(* CoDeSys 2.3.9.41 project: Main.pro *)
(* Libraries: STANDARD.LIB 4.10.05 11:14:46, IECSFC.LIB 13.4.06 15:51:28, ANALYZATION.LIB 5.10.99 09:05:06, Util.lib 18.5.10 15:14:28 *)

(* PLC configuration (modules and I/O channels)
I0 AT %IX0.0 [BitInput] Discrete input 1 {ChannellName = Enter name}
I1 AT %IX0.1 [BitInput] Discrete input 2 {ChannellName = Enter name}
I2 AT %IX0.2 [BitInput] Discrete input 3 {ChannellName = Enter name}
I3 AT %IX0.3 [BitInput] Discrete input 4 {ChannellName = Enter name}
AT %IB1.0 [ByteInput] 8 discrete inputs {ChannellName = Enter name}
AT %IB1.1 [ByteInput] 4 discrete inputs {ChannellName = Enter name}
Q0 AT %QX2.0 [BitOutput] Fast discrete output 1 {ChannellName = Enter name}
AT %QX2.1 [BitOutput] Fast discrete output 2 {ChannellName = Enter name}
AT %QX2.2 [BitOutput] Fast discrete output 3 {ChannellName = Enter name}
AT %QX2.3 [BitOutput] Fast discrete output 4 {ChannellName = Enter name}
AT %QB3.0 [ByteOutput] 8 discrete outputs {ChannellName = Enter name}
AT %QB3.1 [ByteOutput] 8 discrete outputs {ChannellName = Enter name}
AT %IR4.0 [FloatInputP] You need to reboot PLC after change AI configuration! {ChannellName = Fast analog input; AIN_TYPE = 4-20 mA; Peak_Filtr = 200; Flt_Ch = Off; TauRC = 10; MinFV = 0; MaxFV = 20000.0}
AT %IR4.1 [FloatInputP] You need to reboot PLC after change AI configuration! {ChannellName = Fast analog input; AIN_TYPE = 4-20 mA; Peak_Filtr = 200; Flt_Ch = Off; TauRC = 10; MinFV = 0; MaxFV = 20000.0}
AT %IR4.2 [FloatInputP] You need to reboot PLC after change AI configuration! {ChannellName = Fast analog input; AIN_TYPE = 4-20 mA; Peak_Filtr = 200; Flt_Ch = Off; TauRC = 10; MinFV = 0; MaxFV = 20000.0}
AT %IR4.3 [FloatInputP] You need to reboot PLC after change AI configuration! {ChannellName = Fast analog input; AIN_TYPE = 4-20 mA; Peak_Filtr = 200; Flt_Ch = Off; TauRC = 10; MinFV = 0; MaxFV = 20000.0}
AT %IR4.4 [FloatInputP] You need to reboot PLC after change AI configuration! {ChannellName = Fast analog input; AIN_TYPE = 4-20 mA; Peak_Filtr = 200; Flt_Ch = Off; TauRC = 10; MinFV = 0; MaxFV = 20000.0}
AT %IR4.5 [FloatInputP] You need to reboot PLC after change AI configuration! {ChannellName = Fast analog input; AIN_TYPE = 4-20 mA; Peak_Filtr = 200; Flt_Ch = Off; TauRC = 10; MinFV = 0; MaxFV = 20000.0}
AT %IR4.6 [FloatInputP] You need to reboot PLC after change AI configuration! {ChannellName = Fast analog input; AIN_TYPE = 4-20 mA; Peak_Filtr = 200; Flt_Ch = Off; TauRC = 10; MinFV = 0; MaxFV = 20000.0}
AT %IR4.7 [FloatInputP] You need to reboot PLC after change AI configuration! {ChannellName = Fast analog input; AIN_TYPE = 4-20 mA; Peak_Filtr = 200; Flt_Ch = Off; TauRC = 10; MinFV = 0; MaxFV = 20000.0}
AT %IW4.8 [WordInput] AI read time (10ms) {ChannellName = Enter name}
Analog outputs [ID126] node 5, in %IB5 out %QB5 {ChannellName = Analog outputs}
  AT %QR5.0 [FloatOutputP] AO #1 {ChannellName = Analog output; AOUT_TYPE = 4-20 mA; SafeValueREAL = 0.0}
  AT %QR5.1 [FloatOutputP] AO #2 {ChannellName = Analog output; AOUT_TYPE = 4-20 mA; SafeValueREAL = 0.0}
  AT %QR5.2 [FloatOutputP] AO #3 {ChannellName = Analog output; AOUT_TYPE = 4-20 mA; SafeValueREAL = 0.0}
  AT %QR5.3 [FloatOutputP] AO #4 {ChannellName = Analog output; AOUT_TYPE = 4-20 mA; SafeValueREAL = 0.0}
Special input [ID103] node 6, in %IB6 out %QB6 {ChannellName = Special input}
  AT %IX6.0 [BitInput] Special input {ChannellName = Enter name}
Special output [ID104] node 7, in %IB7 out %QB7 {ChannellName = Special output}
  AT %QX7.0 [BitOutput] Special output {ChannellName = Enter name}
*)

(* POU PLC_PRG, FBD *)
PROGRAM PLC_PRG
VAR
	START: BOOL:= FALSE;
	DEC_TO_BIN: DEC_TO_BIN;
	START_RS: RS;
	DTB: DEC_TO_BIN;
	SEND: BOOL := FALSE;
	POSITION: DWORD;
	SENDING: BOOL;
	SENDING_TIMER: TOF;
	INSTRUCTION: ARRAY [1..7] OF DWORD:= 0,14,17,15,7,9,7 11,12,10, 7, 3, 4, 2, 18, 21, 19, 7, 9, 7, 11,12,10, 7, 3, 4, 2, 22, 25, 23, 7, 9, 7, 11,12,10, 7, 3, 4, 2, 26, 29, 27, 7, 9, 7, 11,12,10, 7, 3, 4, 2, 0;
	POSITION_INDEX: INT:=1;

	RESET: BOOL;
END_VAR
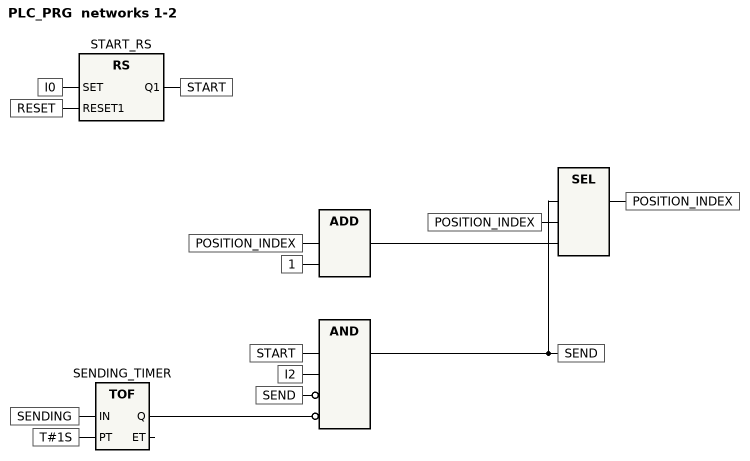
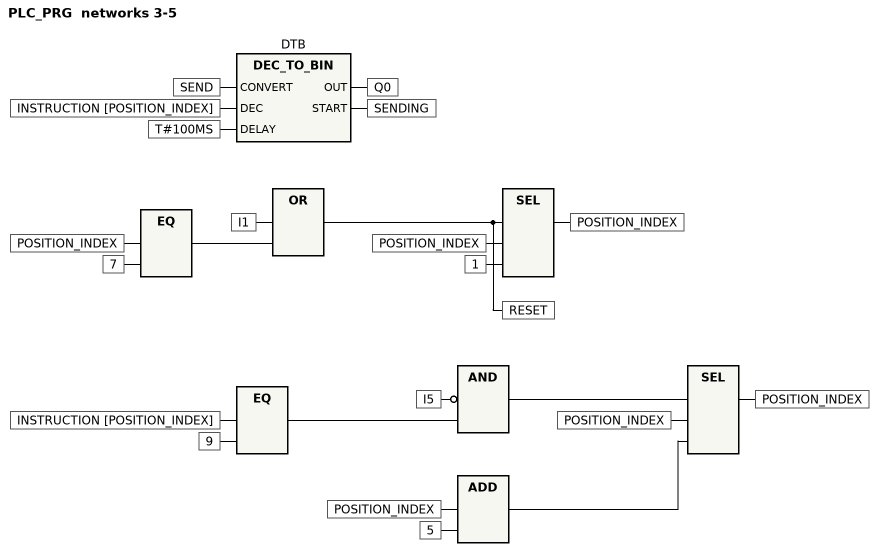
_FBD_ (* Function Block Diagram *)
NETWORK 1
	START_RS:RS(SET: I0, RESET1: RESET) => START
NETWORK 2
	SEL(<AND(START, I2, NOT SEND, NOT SENDING_TIMER:TOF(IN: SENDING, PT: T#1S)) => SEND>, POSITION_INDEX, ADD(POSITION_INDEX, 1)) => POSITION_INDEX
NETWORK 3
	DTB:DEC_TO_BIN(CONVERT: SEND, DEC: INSTRUCTION [POSITION_INDEX], DELAY: T#100MS, START => SENDING) => Q0
NETWORK 4
	SEL(<OR(I1, EQ(POSITION_INDEX, 7)) => RESET>, POSITION_INDEX, 1) => POSITION_INDEX
NETWORK 5
	SEL(AND(NOT I5, EQ(INSTRUCTION [POSITION_INDEX], 9)), POSITION_INDEX, ADD(POSITION_INDEX, 5)) => POSITION_INDEX
_END_FBD_
(* the same logic as Structured Text *)
(* Network 1 *)
START_RS(SET := I0, RESET1 := RESET);
START := START_RS.Q1;
(* Network 2 *)
SENDING_TIMER(IN := SENDING, PT := T#1S);
SEND := START AND I2 AND NOT SEND AND NOT SENDING_TIMER.Q;
POSITION_INDEX := SEL(SEND, POSITION_INDEX, POSITION_INDEX + 1);
(* Network 3 *)
DTB(CONVERT := SEND, DEC := INSTRUCTION [POSITION_INDEX], DELAY := T#100MS);
SENDING := DTB.START;
Q0 := DTB.OUT;
(* Network 4 *)
RESET := I1 OR (POSITION_INDEX = 7);
POSITION_INDEX := SEL(RESET, POSITION_INDEX, 1);
(* Network 5 *)
POSITION_INDEX := SEL(NOT I5 AND ((INSTRUCTION [POSITION_INDEX]) = 9), POSITION_INDEX, POSITION_INDEX + 5);
END_PROGRAM

(* POU DEC_TO_BIN, FBD *)
FUNCTION_BLOCK DEC_TO_BIN
VAR_INPUT
	CONVERT :BOOL :=FALSE;
	DEC :DWORD := 0;
	DELAY: TIME:= T#100MS;
END_VAR
VAR_OUTPUT
	OUT : BOOL :=FALSE;
	START : BOOL :=FALSE;
END_VAR
VAR
	RESET: BOOL :=FALSE;
	Q0, Q1,Q2,Q3,Q4,Q5,Q6,Q7,Q8,Q9,Q10: BOOL :=FALSE;
	TIMER0: TON;
	B, B0, B1,B2,B3: BOOL :=FALSE;
	TIMER6: TON;
	SETTER: RS;
	TIMER: TON;
	SETTER1: RS;
	SETTER0: RS;
	SETTER2: RS;
	SETTER3: RS;
	SETTER4: RS;
	TIMER1: TON;
	TIMER2: TON;
	TIMER3: TON;
	TIMER4: TON;
	RESET0: RS;
	TIMER5: TON;
	TIMER7: TON;
	TIMER8: TON;
	TIMER9: TON;
END_VAR
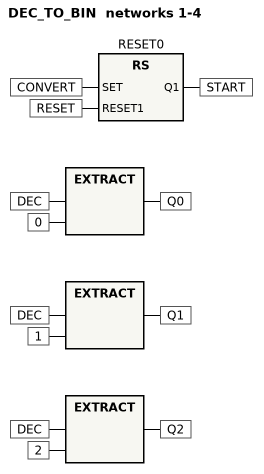
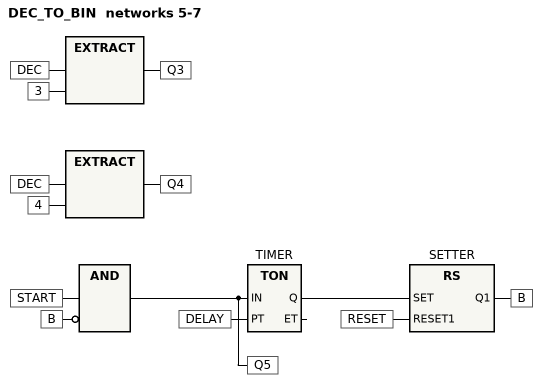
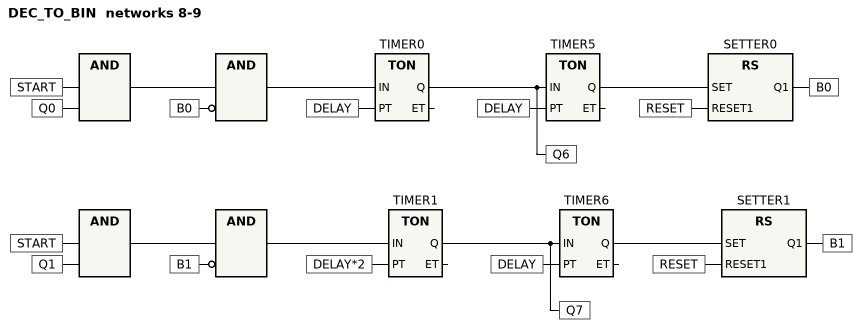
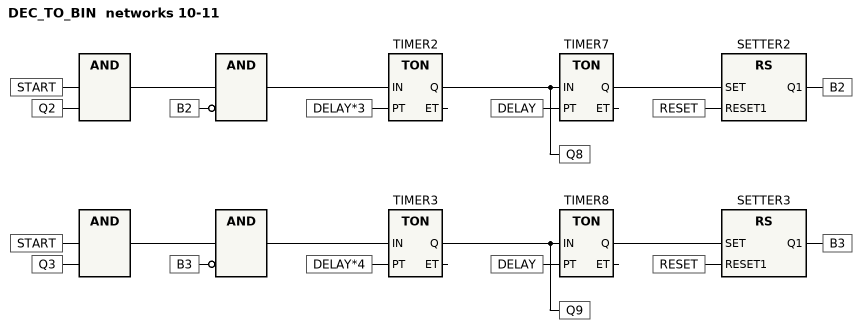
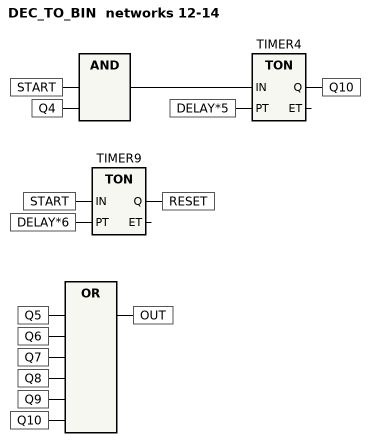
_FBD_ (* Function Block Diagram *)
NETWORK 1
	RESET0:RS(SET: CONVERT, RESET1: RESET) => START
NETWORK 2
	EXTRACT(DEC, 0) => Q0
NETWORK 3
	EXTRACT(DEC, 1) => Q1
NETWORK 4
	EXTRACT(DEC, 2) => Q2
NETWORK 5
	EXTRACT(DEC, 3) => Q3
NETWORK 6
	EXTRACT(DEC, 4) => Q4
NETWORK 7
	SETTER:RS(SET: TIMER:TON(IN: <AND(START, NOT B) => Q5>, PT: DELAY), RESET1: RESET) => B
NETWORK 8
	SETTER0:RS(SET: TIMER5:TON(IN: <TIMER0:TON(IN: AND(AND(START, Q0), NOT B0), PT: DELAY) => Q6>, PT: DELAY), RESET1: RESET) => B0
NETWORK 9
	SETTER1:RS(SET: TIMER6:TON(IN: <TIMER1:TON(IN: AND(AND(START, Q1), NOT B1), PT: DELAY*2) => Q7>, PT: DELAY), RESET1: RESET) => B1
NETWORK 10
	SETTER2:RS(SET: TIMER7:TON(IN: <TIMER2:TON(IN: AND(AND(START, Q2), NOT B2), PT: DELAY*3) => Q8>, PT: DELAY), RESET1: RESET) => B2
NETWORK 11
	SETTER3:RS(SET: TIMER8:TON(IN: <TIMER3:TON(IN: AND(AND(START, Q3), NOT B3), PT: DELAY*4) => Q9>, PT: DELAY), RESET1: RESET) => B3
NETWORK 12
	TIMER4:TON(IN: AND(START, Q4), PT: DELAY*5) => Q10
NETWORK 13
	TIMER9:TON(IN: START, PT: DELAY*6) => RESET
NETWORK 14
	OR(Q5, Q6, Q7, Q8, Q9, Q10) => OUT
_END_FBD_
(* the same logic as Structured Text *)
(* Network 1 *)
RESET0(SET := CONVERT, RESET1 := RESET);
START := RESET0.Q1;
(* Network 2 *)
Q0 := EXTRACT(DEC, 0);
(* Network 3 *)
Q1 := EXTRACT(DEC, 1);
(* Network 4 *)
Q2 := EXTRACT(DEC, 2);
(* Network 5 *)
Q3 := EXTRACT(DEC, 3);
(* Network 6 *)
Q4 := EXTRACT(DEC, 4);
(* Network 7: see the listing above *)
(* Network 8 *)
TIMER0(IN := (START AND Q0) AND NOT B0, PT := DELAY);
Q6 := TIMER0.Q;
TIMER5(IN := TIMER0.Q, PT := DELAY);
SETTER0(SET := TIMER5.Q, RESET1 := RESET);
B0 := SETTER0.Q1;
(* Network 9 *)
TIMER1(IN := (START AND Q1) AND NOT B1, PT := DELAY*2);
Q7 := TIMER1.Q;
TIMER6(IN := TIMER1.Q, PT := DELAY);
SETTER1(SET := TIMER6.Q, RESET1 := RESET);
B1 := SETTER1.Q1;
(* Network 10 *)
TIMER2(IN := (START AND Q2) AND NOT B2, PT := DELAY*3);
Q8 := TIMER2.Q;
TIMER7(IN := TIMER2.Q, PT := DELAY);
SETTER2(SET := TIMER7.Q, RESET1 := RESET);
B2 := SETTER2.Q1;
(* Network 11 *)
TIMER3(IN := (START AND Q3) AND NOT B3, PT := DELAY*4);
Q9 := TIMER3.Q;
TIMER8(IN := TIMER3.Q, PT := DELAY);
SETTER3(SET := TIMER8.Q, RESET1 := RESET);
B3 := SETTER3.Q1;
(* Network 12 *)
TIMER4(IN := START AND Q4, PT := DELAY*5);
Q10 := TIMER4.Q;
(* Network 13 *)
TIMER9(IN := START, PT := DELAY*6);
RESET := TIMER9.Q;
(* Network 14 *)
OUT := Q5 OR Q6 OR Q7 OR Q8 OR Q9 OR Q10;
END_FUNCTION_BLOCK
